// TwinCAT 3 PLC project PLC_SerialCom_Sample1
// ProgramVersion: 3.1.0.8
// libraries:
//   Tc2_SerialCom, * (Beckhoff Automation GmbH)
//   Tc2_Standard, * (Beckhoff Automation GmbH)
//   Tc3_Module, * (Beckhoff Automation GmbH)
// project tree:
//   GVLs/ GVL.TcGVL
//   / PlcTask_Fast.TcTTO (not stored), PlcTask_Standard.TcTTO (not stored)
//   POUs/ Background.TcPOU, BackgroundKL.TcPOU, BackgroundEL.TcPOU (not stored), FB_SerialCom.TcPOU, MAIN.TcPOU, BackgroundPcCOM.TcPOU (not stored)
// real-time tasks:
//   TASK PlcTask_Fast: cycle T#2ms, priority 19, ADS port 350
//   TASK PlcTask_Standard: cycle T#10ms, priority 20, ADS port 351
// I/O:
//   DEVICE Device 1 (COM Port)
//   DEVICE Device 3 (EtherCAT) (disabled), AmsNetId 172.17.60.154.4.1
//     Term 1 (EK1100) [EK1100 EtherCAT Coupler (2A E-Bus)]
//       Term 2 (EL6001) [EL6001 Interface (RS232)]
//       Box 3 (BK1250)
//   DEVICE Device 2 (EtherCAT), AmsNetId 5.109.45.144.3.1
// variable links:
//   PLC_SerialCom_Sample1/PLC_SerialCom_Sample1 Instance <-> Device 1 (COM Port)
//     PlcTask_Standard Inputs/BackgroundPcCOM.stIn_PcCom/D <-> Inputs/Data1
//     PlcTask_Standard Inputs/BackgroundPcCOM.stIn_PcCom/D @bit {8..504 step 8} <-> Inputs/Data{2..64}  (63 links)
//     PlcTask_Standard Inputs/BackgroundPcCOM.stIn_PcCom/SerStatus <-> Inputs/Status
//     PlcTask_Standard Outputs/BackgroundPcCOM.stOut_PcCom/D <-> Outputs/Data1
//     PlcTask_Standard Outputs/BackgroundPcCOM.stOut_PcCom/D @bit {8..504 step 8} <-> Outputs/Data{2..64}  (63 links)
//     PlcTask_Standard Outputs/BackgroundPcCOM.stOut_PcCom/SerCtrl <-> Outputs/Ctrl
//   PLC_SerialCom_Sample1/PLC_SerialCom_Sample1 Instance <-> Device 3 (EtherCAT)/Term 1 (EK1100)/Box 3 (BK1250)
//     PlcTask_Fast Inputs/BackgroundKL.stIn_KL6001/D[0] <-> Term 3 (KL6001-A)/Channel 1/Data In 0
//     PlcTask_Fast Inputs/BackgroundKL.stIn_KL6001/D[1] <-> Term 3 (KL6001-A)/Channel 1/Data In 1
//     PlcTask_Fast Inputs/BackgroundKL.stIn_KL6001/D[2] <-> Term 3 (KL6001-A)/Channel 1/Data In 2
//     PlcTask_Fast Inputs/BackgroundKL.stIn_KL6001/SerStatus <-> Term 3 (KL6001-A)/Channel 1/Ser. State
//     PlcTask_Fast Inputs/BackgroundKL.stIn_KL6001/Status <-> Term 3 (KL6001-A)/Channel 1/State
//     PlcTask_Fast Outputs/BackgroundKL.stOut_KL6001/Ctrl <-> Term 3 (KL6001-A)/Channel 1/Ctrl
//     PlcTask_Fast Outputs/BackgroundKL.stOut_KL6001/D[0] <-> Term 3 (KL6001-A)/Channel 1/Data Out 0
//     PlcTask_Fast Outputs/BackgroundKL.stOut_KL6001/D[1] <-> Term 3 (KL6001-A)/Channel 1/Data Out 1
//     PlcTask_Fast Outputs/BackgroundKL.stOut_KL6001/D[2] <-> Term 3 (KL6001-A)/Channel 1/Data Out 2
//     PlcTask_Fast Outputs/BackgroundKL.stOut_KL6001/SerCtrl <-> Term 3 (KL6001-A)/Channel 1/Ser. Ctrl
//   PLC_SerialCom_Sample1/PLC_SerialCom_Sample1 Instance <-> Device 3 (EtherCAT)/Term 1 (EK1100)/Term 2 (EL6001)
//     PlcTask_Fast Inputs/BackgroundEL.stIn_EL6001/D <-> Inputs/Data In 0
//     PlcTask_Fast Inputs/BackgroundEL.stIn_EL6001/D @bit {8..168 step 8} <-> Inputs/Data In {1..21}  (21 links)
//     PlcTask_Fast Inputs/BackgroundEL.stIn_EL6001/Status <-> Inputs/Status
//     PlcTask_Fast Outputs/BackgroundEL.stOut_EL6001/Ctrl <-> Outputs/Ctrl
//     PlcTask_Fast Outputs/BackgroundEL.stOut_EL6001/D <-> Outputs/Data Out 0
//     PlcTask_Fast Outputs/BackgroundEL.stOut_EL6001/D @bit {8..168 step 8} <-> Outputs/Data Out {1..21}  (21 links)

// ---- GVLs/GVL.TcGVL
VAR_GLOBAL
	RxBufferEL			: ComBuffer;	(* Receive data buffer; used with all receive function blocks *)
	TxBufferEL			: ComBuffer;	(* Transmit data buffer; used with all receive function blocks *)

	RxBufferKL			: ComBuffer;	(* Receive data buffer; used with all receive function blocks *)
	TxBufferKL			: ComBuffer;	(* Transmit data buffer; used with all receive function blocks *)
END_VAR

// ---- POUs/Background.TcPOU
PROGRAM Background
VAR
END_VAR

(*
The SerialLineControl function block is supposed to be called in every PLC cycle.
It communicates with the serial line hardware device and transmits or receives data.
The SerialLineControl can be called in the standard task (e.g.for PcCOM port usage) 
or in a separate fast task (e.g.for terminal usage) as well.
A fast separate task will be necessary at high baud rates or with KL6001 terminals 
which have a small process image (3 or 5 data bytes only)
*)

(* background communication with the EL6001 terminal *)
BackgroundEL();

(* background communication with the KL6001 terminal (3byte) *)
BackgroundKL();

END_PROGRAM

// ---- POUs/BackgroundKL.TcPOU
PROGRAM BackgroundKL
VAR
	(* background communication with the KL6001 terminal (3byte) *)
	fbKL6001Ctrl		: SerialLineControl;
	bKL6001CtrlError	: BOOL;
	eKL6001CtrlErrorID	: ComError_t;
	fbKL6001Config		: KL6configuration;
	bKL6001ConfigError	: BOOL;
	eKL6001ConfigErrorID: ComError_t;
	bKL6001ConfigExe	: BOOL := TRUE;
	(* 	I/O variables for a KL6001 terminal*)
	stIn_KL6001 AT %I*	: KL6inData;	(* linked to the KL6001 in the TwinCAT System Manager *)
	stOut_KL6001 AT %Q*	: KL6outData;	(* linked to the KL6001 in the TwinCAT System Manager *)
END_VAR

(*
The SerialLineControl function block is supposed to be called in every PLC cycle.
It communicates with the serial line hardware device and transmits or receives data.
The SerialLineControl can be called in the standard task (e.g.for PcCOM port usage) 
or in a separate fast task (e.g.for terminal usage) as well.
A fast separate task will be necessary at high baud rates or with KL6001 terminals 
which have a small process image (3 or 5 data bytes only)
*)

(* background communication with the KL6001 terminal (3byte) *)
fbKL6001Config(
	Execute:= bKL6001ConfigExe, 
	Mode:= SERIALLINEMODE_KL6_3B_ALTERNATIVE, 
	Baudrate:= 9600, 
	NoDatabits:= 8, 
	Parity:= 0, 
	Stopbits:= 1, 
	Handshake:= HANDSHAKE_NONE, 
	ContinousMode:= FALSE, 
	pComIn:= ADR(stIn_KL6001), 
	pComOut:= ADR(stOut_KL6001), 
	SizeComIn:= SIZEOF(stIn_KL6001), 
	Done=> , 
	Busy=> , 
	Error=> , 
	ErrorId=>  );
IF fbKL6001Config.Error THEN
	bKL6001ConfigError := TRUE;
	eKL6001ConfigErrorID := fbKL6001Config.ErrorId;
END_IF
	
IF NOT fbKL6001Config.Busy AND NOT bKL6001ConfigError THEN
	bKL6001ConfigExe := FALSE;
	fbKL6001Ctrl(
		Mode:= SERIALLINEMODE_KL6_3B_ALTERNATIVE,
		pComIn:= ADR(stIn_KL6001),
		pComOut:= ADR(stOut_KL6001),
		SizeComIn:= SIZEOF(stIn_KL6001),
		Error=> ,
		ErrorID=> ,
		TxBuffer:= TxBufferKL,
		RxBuffer:= RxBufferKL );
	IF fbKL6001Ctrl.Error THEN
		bKL6001CtrlError := TRUE;
		eKL6001CtrlErrorID := fbKL6001Ctrl.ErrorID;
	END_IF
END_IF

END_PROGRAM

// ---- POUs/FB_SerialCom.TcPOU
FUNCTION_BLOCK FB_SerialCom
VAR_IN_OUT
	TxBuffer	: ComBuffer;
	RxBuffer	: ComBuffer;
END_VAR
VAR
	Timer		: TON := (PT:=T#1S);
	fbSend		: SendString;
	bSendBusy	: BOOL;
	eSendErrorID: ComError_t;

	fbReceive		: ReceiveString;
	sReceivedString	: STRING;
	sLastReceivedString: STRING;
	bStringReceived	: BOOL;
	bReceiveBusy	: BOOL;
	bReceiveError	: BOOL;
	eReceiveErrorID	: ComError_t;
	bReceiveTimeout	: BOOL;
	nReceiveCounter	: UDINT;
END_VAR

// Call the send block every second to repeat the transmission.
// Also call the block as long as it is busy to finish a transmission.
Timer(IN:=TRUE);
IF Timer.Q OR fbSend.Busy THEN
	Timer(IN:=FALSE); (* reset timer *)
	fbSend(	SendString:= '$02Hello World ! $03',
			TXbuffer:= TxBuffer,
			Busy=> bSendBusy,
			Error=> );
	IF fbSend.Error <> COMERROR_NOERROR THEN
		eSendErrorID := fbSend.Error;
	END_IF
END_IF

//	Receive string data:
//	The block receives any data strings beginning with a STX ($02) and ending with an ETX ($03) character.	
fbReceive(
	Prefix:= '$02',
	Suffix:= '$03',
	Timeout:= T#1s,
	ReceivedString:= sReceivedString,
	RXbuffer:= RxBuffer,
	StringReceived=> bStringReceived,
	Busy=> bReceiveBusy,
	Error=> ,
	RxTimeout=> bReceiveTimeout );
IF fbReceive.Error <> COMERROR_NOERROR THEN
	eReceiveErrorID := fbReceive.Error;
END_IF
IF bStringReceived THEN
	nReceiveCounter := nReceiveCounter + 1;
	sLastReceivedString := sReceivedString;
END_IF

END_FUNCTION_BLOCK

// ---- POUs/MAIN.TcPOU
(*
SerialCom_InfoSys_Sample1 (v2.0)
This sample sends and receives a string via serial communication.
Three hardware interfaces are used: Pc COM port, EL terminal, KL terminal
*)
PROGRAM MAIN
VAR
	fbPcCom		: FB_SerialCom;
	fbEL6001	: FB_SerialCom;
	fbKL6001	: FB_SerialCom;
	
	(* exchange buffers with background communication with the PC COM port device *)
	RxBufferPcCom	: ComBuffer;	(* Receive data buffer; used with all receive function blocks *)
	TxBufferPcCom	: ComBuffer;	(* Transmit data buffer; used with all receive function blocks *)
END_VAR


(* background communication with the PC COM port device *)
BackgroundPcCOM(RxBufferPcCom:=RxBufferPcCom, TxBufferPcCom:=TxBufferPcCom);


(* Send and receive commands *)
fbPcCom(TxBuffer:=TxBufferPcCom, RxBuffer:=RxBufferPcCom);

fbEL6001(TxBuffer:=TxBufferEL, RxBuffer:=RxBufferEL);

fbKL6001(TxBuffer:=TxBufferKL, RxBuffer:=RxBufferKL);

END_PROGRAM
